(* CODESYS project stec.project

Project tree, tasks and I/O mapping:
  Device : CODESYS Control Win V3, 3S - Smart Software Solutions GmbH, order no. 305021, version 3.5.6.10
    application Application
      libraries: Standard, * (System); Util, * (System)
      task CLP (cyclic, interval t#500ms, priority 1) calls CLP_CONF700
      task executaprocesso (cyclic, interval t#500ms, priority 1) calls Processo
      task RedeFF (cyclic, interval t#500ms, priority 1) calls LD_LT1, LD_LT2, LD_FT1, LD_FT2, LD_FT3, LD_FT4, TT302, FI_01, FI_02
      program CLP_CONF700 [LD]
      global variables CLP_entrada
      global variables CLP_saida
      global variables Var_processo
      function block AI [FBD]
      function block AO [FBD]
      function block PIDCONTROL [FBD]
      program LD_LT1 [FBD]
      function block ALARME [LD]
      program Processo [ST]
      Symbols
      program LD_LT2 [FBD]
      program LD_FT1 [FBD]
      program LD_FT2 [FBD]
      program LD_FT3 [FBD]
      program LD_FT4 [FBD]
      program FI_01 [FBD]
      program TT302 [FBD]
      program FI_02 [FBD]
      global variables Par_processo
      function block ControladorPID [ST]
*)

// Device/Application/CLP_entrada
VAR_GLOBAL
HI_LEVEL01	:BOOL;   // indicação de nivel alto no TAQ
HI_LEVEL02	:BOOL;   // indicação de nivel alto no TP
HI_TEMP01	:BOOL;   // indicação de temperatura alta no TAQ
HI_TEMP02	:BOOL;   // indicação de temperatura altra no TP
HI_FLOW01	:BOOL;   // Indicação de vazão alta na saída do TP
LO_LEVEL01	:BOOL;   // indicação de nivel baixo no TAQ
LO_LEVEL02	:BOOL;   //indicação de nivel baixo no TP

// considere que 01 é TAQ e 02 é TP
END_VAR

// Device/Application/CLP_saida
VAR_GLOBAL
B02	:BOOL;  //comando para ligar/desligar a bomba 1  entrada TP e TAQ
B01	:BOOL;  //comando para ligar/desligar a bomba 2 saida TP
RES	:BOOL;  // comando para ligar/desligar a resistência
END_VAR

// Device/Application/Var_processo
VAR_GLOBAL
	// variáveis anaógicas de saída do processo
	L_TAQ  :REAL :=0.0;  // nivel do TAQ : LT01
	L_TP   :REAL :=0.0;   // nivel do TP : LT02
	T_TAQ  :REAL :=23.5;  // temperatura medida no TAQ :TT01
	T_TP   :REAL :=23.5;   // Temperatura medida no TP : TT02
	Temp_TAQ  :REAL :=23.5;  // temperatura real no TAQ :TT01
	Temp_TP   :REAL :=23.5;   // Temperatura real no TP : TT02
	FI_TAQ :REAL:=0.0;   // Vazão de entrada do TAQ : FT01
	FO_TAQ :REAL:=0.0;   // Vazão saida do TAQ  :FT02
	FI_TP :REAL:=0.0;   // Vazão de entrada do TP : FT03
	FO_TP :REAL:=0.0;   // Vazão saida do TP : FT04
	// variáveis anológicas de entrada do processo
	VI_TAQ :REAL;  // comando para vávula FV01 (LCV1) entrada do TAQ 
	VO_TAQ :REAL;  // comando para vávula FV02 (TCV1) saida do TAQ
    VI_TP :REAL;   // comando para vávula FV03 (LCV2) entrada do TP
	VO_TP :REAL;  // comando para vávula FV04 (FCV1) saida do TP
	TC_TAQ : REAL; // comando para resistência de aquecimento do TAQ (TTC01)
	// variáveis de interface com o CLP
	
END_VAR

// Device/Application/Par_processo
VAR_GLOBAL
	// valores de parametrização do nivel do TAQ
LTAQMAX: REAL := 500.0; // Nível máximo do TAQ
LTAQMIN: REAL :=0.0;   // Nivel minimo do TAQ
LSHTAQ:REAL :=450.0;  // Limite para alarme de nível alto
LSLTAQ:REAL :=60.0;   // Limite para alarme de nível baixo

	//valores de parametrização do nivel do TP
LTPMAX: REAL := 700.0; // Nível máximo do TP
LTPMIN: REAL :=0.0;   // Nivel minimo do TP
LSHTP:REAL :=650.0;  // Limite para alarme de nível alto
LSLTP:REAL :=50.0;   // Limite para alarme de nível baixo

//valores de parametrização da tempearatura do TAQ
TSHTAQ:REAL :=80.0;  // Limite para alarme de temperatura alta alto
TTPMAX: REAL := 100.0;//Temperatura máxima para o TP
TTPMIN: REAL :=0.0;   // Temperatura minima para o TP

//valores de parametrização da tempearatura do TP
TTAQMAX: REAL := 100.0;//Temperatura máxima para o TAQ
TTAQMIN: REAL :=0.0;   // Temperatura minima para o TAQ
TSHTP:REAL :=50.0;  // Limite para alarme de temperatura alta alto

//valores de parametrização da vazao entrada TAQ
FIXTAQ :REAL :=44.0;   // vazão máxima de entrada do TAQ
FIITAQ :REAL :=0.0;     // vazão mínima de entrada do TAQ

//valores de parametrização da vazão saida TAQ
FOXTAQ :REAL :=9.0;   // vazão máxima de saida do TAQ
FOITAQ :REAL :=0.0;     // vazão mínima de saida do TAQ

//valores de parametrização da vazão entrada TP
FIXTP :REAL :=34.0;   // vazão máxima de entrada do TP
FIITP :REAL :=0.0;     // vazão mínima de entrada do TP

//valores de parametrização da vazão saida TP
FOXTP :REAL :=56.0;   // vazão máxima de saida do TP
FOITP :REAL :=0.0;    // vazão mínima de saida do TP
FSH4:REAL :=57.0;  // Limite para alarme de nível alto


//valores de parametrização da potência da resistência de aquecimento do TAQ
PMAX:REAL:=12000;
Temp_Reservatorio:REAL:=23;

DELTAT:REAL:=0.5;     // intervalode de amostragem deve corresponder ao tempo de ciclo da tarefa

END_VAR

// Device/Application/CLP_CONF700
PROGRAM CLP_CONF700
VAR
 
SHB02	:BOOL;   // cahve de software via SCADA para ligar a bomba 2
SHB01	:BOOL;   // cahve de software via SCADA para ligar a bomba 1
SHRES	:BOOL;   // cahve de software via SCADA para ligar a resistência
END_VAR

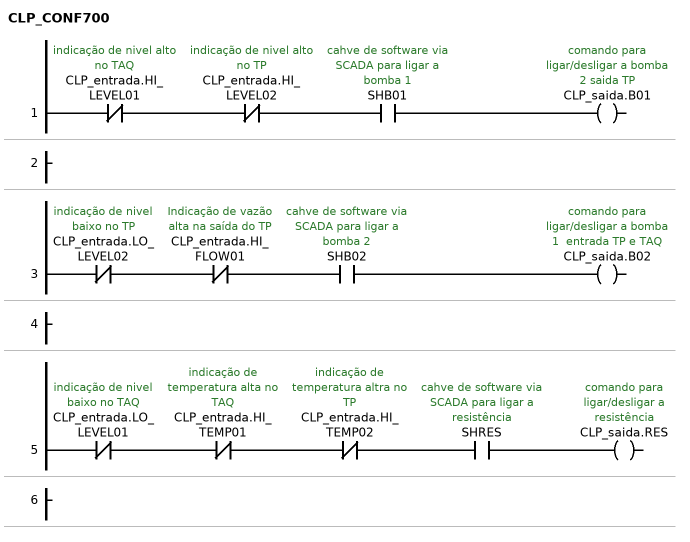
// NETWORK 1
//   CLP_entrada.HI_LEVEL01: indicação de nivel alto no TAQ
//   CLP_entrada.HI_LEVEL02: indicação de nivel alto no TP
//   SHB01: cahve de software via SCADA para ligar a bomba 1
//   CLP_saida.B01: comando para ligar/desligar a bomba 2 saida TP
CLP_saida.B01 := NOT CLP_entrada.HI_LEVEL01 AND NOT CLP_entrada.HI_LEVEL02 AND SHB01;

// NETWORK 2

// NETWORK 3
//   CLP_entrada.LO_LEVEL02: indicação de nivel baixo no TP
//   CLP_entrada.HI_FLOW01: Indicação de vazão alta na saída do TP
//   SHB02: cahve de software via SCADA para ligar a bomba 2
//   CLP_saida.B02: comando para ligar/desligar a bomba 1 entrada TP e TAQ
CLP_saida.B02 := NOT CLP_entrada.LO_LEVEL02 AND NOT CLP_entrada.HI_FLOW01 AND SHB02;

// NETWORK 4

// NETWORK 5
//   CLP_entrada.LO_LEVEL01: indicação de nivel baixo no TAQ
//   CLP_entrada.HI_TEMP01: indicação de temperatura alta no TAQ
//   CLP_entrada.HI_TEMP02: indicação de temperatura altra no TP
//   SHRES: cahve de software via SCADA para ligar a resistência
//   CLP_saida.RES: comando para ligar/desligar a resistência
CLP_saida.RES := NOT CLP_entrada.LO_LEVEL01 AND NOT CLP_entrada.HI_TEMP01 AND NOT CLP_entrada.HI_TEMP02 AND SHRES;

// NETWORK 6

END_PROGRAM

// Device/Application/Processo
PROGRAM Processo
VAR
BETA:REAL:=0.7;   // valor do filtro das vazões
offset:REAL:=23.4;  //  temperatura inicial
cont:INT;         //contador de atrasos
// parametros vazão entrada ATQ
KITAQ:REAL :=  0.73;        // ganho vazão entrada TAQ
ATITAQ:REAL := 4.0;     //  atraso em segundos vazão entrada TAQ
VIATAQ : ARRAY [1..10] OF REAL := [0,0,0,0,0,0,0,0,0,0];  // vetor com valores anteriores da valvula de entrada TAQ
FIATAQ : REAL;  // valor anterior da vazaão de entrada TAQ
KOTAQ:REAL :=  0.128;        // ganho vazão saida TAQ
ATOTAQ:REAL := 4.0;     //  atraso em segundos vazão saida TAQ
VOATAQ : ARRAY [1..10] OF REAL := [0,0,0,0,0,0,0,0,0,0];  // vetor com valores anteriores da valvula saida TAQ
FOATAQ : REAL;  // valor anterior da vazaão de saida TAQ
// parametro para as vazões do TP

KITP:REAL :=  0.68;        // ganho vazão entrada TP
ATITP:REAL := 4.0;     //  atraso em segundos vazão entrada TP
VIATP : ARRAY [1..10] OF REAL := [0,0,0,0,0,0,0,0,0,0];  // vetor com valores anteriores da valvula entrada TAQ
FIATP : REAL;  // valor anterior da vazaão de entrada TP
KOTP :REAL := 0.8;  // ganho vazão saida TP
ATOTP:REAL := 3.0;     //  atraso em segundos vazão saida TP
VOATP : ARRAY [1..10] OF REAL := [0,0,0,0,0,0,0,0,0,0];  // vetor com valores anteriores da valvula saida TAQ
FOATP : REAL;  // valor anterior da vazaão de saida TP
VAZAOTP: REAL;  // variável auxiliar para calcula vazao saida TP
// parametro para valvulas do TAQ
VIXTAQ :REAL :=70.0;   // limite superior de saturação para a vazão máxima valvula entrada TAQ
VIITAQ :REAL :=10.0;     // limite inferior de saturação para a vazão máxima valvula entrada TAQ
VOXTAQ :REAL :=90.0;   // limite superior de saturação para a vazão máxima valvula saida TAQ
VOITAQ :REAL :=20.0;     // limite inferior de saturação para a vazão máxima valvula saida TAQ

// parametro para valvulas do TP
VIXTP :REAL :=60.0;   // limite superior de saturação para a vazão máxima valvula entrada TP
VIITP :REAL :=10.0;     // limite inferior de saturação para a vazão máxima valvula entrada TP
VOXTP :REAL :=80.0;   // limite superior de saturação para a vazão máxima valvula saida TP
VOITP :REAL :=10.0;     // limite inferior de saturação para a vazão máxima valvula saida TP

// parametros para caluclo dos nivies
AREA:REAL:=1.140E5;   // Area dos tanques em mm
CONV:REAL:=16.67E3;  //conversaço de l/min para mm3/s
LATAQ:REAL;    // valor anterior do nivel do TAQ
LATP:REAL;    // valor anterior do nivel do TP
VAZAO:REAL;   // variável auxiliar para calculo do balanço da vazão

Temp_TAQ:REAL;
Temp_TP:REAL;
Vol_TP:REAL;
Vol_TAQ:REAL;

//parametros calculo temperatura TAQ

nataq:REAL:=0.9568E-3;   //numerador discreto função de aquecimento do TAQ
dataq:REAL:=-0.999;   //denominador discreto função de aquecimento do TAQ
nftaq:REAL:=0.0102;   //numerador discreto entrada agua fria no TAQ
dftaq:REAL:=-0.9876;   //denominador discreto entrada agua fria no TAQ
uataq:REAL:=0;    // sinal de entrada para aquecimento do TAQ
sataq:REAL:=0;    // parcela da temperatura de aquecimento do TAQ
U1TAQ : ARRAY [1..50] OF REAL := [0,0,0,0,0,0,0,0,0,0,0,0,0,0,0,0,0,0,0,0,0,0,0,0,0,0,0,0,0,0,0,0,0,0,0,0,0,0,0,0,0,0,0,0,0,0,0,0,0,0]; 
uftaq:REAL:=0;    // sinal de entrada para esfriar o  TAQ
sftaq:REAL:=0;    // parcela da temperatura do esfriamento do TAQ
U2TAQ :ARRAY [1..10] OF REAL :=[0,0,0,0,0,0,0,0,0,0];
Ttaq:REAL;    // auxiliar para somar as parcelas da temperatura e saturar entre offset e 100
potencia:REAL:=0; // auxiliar para potencia como liga/desliga da temperatura
antsf:REAL:=0;  //valor anterior da parcela de resfriamento da temperatura
antsa:REAL:=0; // valor anterior da parcela de aquecimento da temperatura
//parametros calculo temperatura TP

natp:REAL:=0.6297E-3;   //numerador discreto função de aquecimento do TP
datp:REAL:=-0.9967;   //denominador discreto função de aquecimento do TP
nftp:REAL:=0.4225E-4;   //numerador discreto entrada agua fria no TP
dftp:REAL:=-0.9850;   //denominador discreto entrada agua fria no TP
uatp:REAL;    // sinal de entrada para aquecimento do TP
satp:REAL;    // parcela da temperatura de aquecimento do TP
U1TP : ARRAY [1..50] OF REAL := [0,0,0,0,0,0,0,0,0,0,0,0,0,0,0,0,0,0,0,0,0,0,0,0,0,0,0,0,0,0,0,0,0,0,0,0,0,0,0,0,0,0,0,0,0,0,0,0,0,0]; 
uftp:REAL;    // sinal de entrada para esfriar o  TP
sftp:REAL;    // parcela da temperatura do esfriamento do TP
U2TP :ARRAY [1..10] OF REAL :=[0,0,0,0,0,0,0,0,0,0];
Ttp:REAL;    // auxiliar para somar as parcelas da temperatura e saturar entre offset e 100
antpsf:REAL:=0;  //valor anterior da parcela de resfriamento da temperatura
antpsa:REAL:=0; // valor anterior da parcela de aquecimento da temperatura
haux, taux, faux:REAL:=0;  // variaveis auxiliaroes
lixo:REAL:=0;
END_VAR

// atualiza os valores anteriores  das vazões
FIATAQ:=Var_processo.FI_TAQ;
FOATAQ:=Var_processo.FO_TAQ;
FIATP:=Var_processo.FI_TP;
FOATP:=Var_processo.FO_TP;
// atualiza os valores anteriores dos niveis
LATAQ:=Var_processo.L_TAQ;
LATP:=Var_processo.L_TP;
// atualiza os valores anteriores das valvulas  e  dos sinais da temperatura
FOR cont:=10 TO 2 BY -1 DO
		VIATAQ[cont]:=VIATAQ[cont-1]; 
		VOATAQ[cont]:=VOATAQ[cont-1]; 
		VIATP[cont]:=VIATP[cont-1]; 
		VOATP[cont]:=VOATP[cont-1]; 
		U2TAQ[cont]:=U2TAQ[cont-1];
		U2TP[cont]:=U2TP[cont-1];
END_FOR
FOR cont:=50 TO 2 BY -1 DO
		U1TAQ[cont]:=U1TAQ[cont-1];
		U1TP[cont]:=U1TP[cont-1];
END_FOR
// garante a saturação das valvulas entre 0 e 100%
IF Var_processo.VI_TAQ < 0.0
	THEN Var_processo.VI_TAQ:=0.0;
END_IF
IF Var_processo.VI_TAQ > 100.0
	THEN Var_processo.VI_TAQ:=100.0;
END_IF

IF Var_processo.VO_TAQ < 0.0
	THEN Var_processo.VO_TAQ:=0.0;
END_IF
IF Var_processo.VO_TAQ > 100.0
	THEN Var_processo.VO_TAQ:=100.0;
END_IF

IF Var_processo.VI_TP < 0.0
	THEN Var_processo.VI_TP:=0.0;
END_IF
IF Var_processo.VI_TP > 100.0
	THEN Var_processo.VI_TP:=100.0;
END_IF

IF Var_processo.VO_TP < 0.0
	THEN Var_processo.VO_TP:=0.0;
END_IF
IF Var_processo.VO_TP > 100.0
	THEN Var_processo.VO_TP:=100.0;
END_IF

// atualiza a posição mais recente dos vetores de atraso das valvulas
VIATAQ[1]:= Var_processo.VI_TAQ;
VOATAQ[1]:= Var_processo.VO_TAQ;
VIATP[1]:= Var_processo.VI_TP;
VOATP[1]:= Var_processo.VO_TP;

// vazão de entrada do TAQ
Var_processo.FI_TAQ:= MIN(0.7*VIATAQ[8],12/(0.5+EXP(-0.125*(VIATAQ[8]-20))));
IF NOT(CLP_saida.B01) // verifica se a bomba está desligada
	THEN Var_processo.FI_TAQ:=0.0;
END_IF
// dinamica da válvula
Var_processo.FI_TAQ:= BETA*Var_processo.FI_TAQ + (1-BETA)*FIATAQ;

// vazão de saida do TAQ
Var_processo.FO_TAQ:=  SQRT(LATAQ/LTAQMAX*2)*MIN(0.2*VOATAQ[8],7.2/(0.8+EXP(-0.1125*(VOATAQ[8]-50)))); 

// dinamica valvula
Var_processo.FO_TAQ:= BETA*Var_processo.FO_TAQ + (1-BETA)*FOATAQ;

// vazão de entrada do TP
Var_processo.FI_TP:=  MIN(1.0*VIATP[8],25.85/(0.615+EXP(-0.1*(VIATP[8]-35))));
IF NOT(CLP_saida.B01) // verifica se a bomba está desligada
	THEN Var_processo.FI_TP:=0.0;
END_IF
 
// coloca um filtro para a mudança não ser muito brusca
Var_processo.FI_TP:= BETA*Var_processo.FI_TP + (1-BETA)*FIATP;

// vazão de saida do TP
//é preciso uma variável auxiliar para evitar que o alarme dispare antes do calculo completo da vazão
VAZAOTP:=  MIN(1.3*VOATP[8],53/(0.964+EXP(-0.097*(VOATP[8]-35))));
IF NOT(CLP_saida.B02) // verifica se a bomba está desligada
	THEN VAZAOTP:=0.0;
END_IF

// dinamica valvula

Var_processo.FO_TP:= BETA*VAZAOTP + (1-BETA)*FOATP;

// calcula os niveis pelo balançco dinamico das vazões
//Nivel do TAQ
VAZAO:=Var_processo.FI_TAQ-Var_processo.FO_TAQ;
VAZAO:=VAZAO*CONV;
Var_processo.L_TAQ:= LATAQ+(VAZAO*DELTAT)/AREA;
IF Var_processo.L_TAQ  < 0.0
	THEN Var_processo.L_TAQ:=0.0;
END_IF
IF Var_processo.L_TAQ > LTAQMAX
	THEN Var_processo.L_TAQ:=LTAQMAX;
END_IF

//Nivel do TP
VAZAO:=Var_processo.FI_TP + Var_processo.FO_TAQ - Var_processo.FO_TP ;
VAZAO:=VAZAO*CONV;
Var_processo.L_TP:= LATP+(VAZAO*DELTAT)/AREA;
IF Var_processo.L_TP  < 0.0
	THEN Var_processo.L_TP:=0.0;
END_IF
IF Var_processo.L_TP > LTPMAX
	THEN Var_processo.L_TP:=LTPMAX;
END_IF

//calculo das temperaturas pelos modelos pelo balanço de massa e energia
//Temperatura do TAQ parcela de aquecimento
IF CLP_saida.RES
	THEN potencia:=Par_processo.PMAX *(Var_processo.TC_TAQ/100+SIN(2*(1-Var_processo.TC_TAQ/100)*3.1416)/(2*3.1416));//(pi-theta)/2 + sin(2theta)/4
	ELSE potencia:=0;
END_IF

Vol_TAQ:=AREA*LATAQ*1E-6+DELTAT*(FIATAQ-FOATAQ)/60;
IF Vol_TAQ<=0
	THEN Vol_TAQ:=1E-2;
END_IF

Temp_TAQ:=Var_processo.Temp_TAQ+potencia*DELTAT/4200/Vol_TAQ;
Temp_TAQ:=Temp_TAQ+FIATAQ*DELTAT/60/Vol_TAQ*(Par_processo.Temp_Reservatorio-Var_processo.Temp_TAQ);

U1TAQ[1]:=Temp_TAQ;   // atualiza a  posição mais recente do vetor de atrasos
Var_processo.T_TAQ := Var_processo.T_TAQ +BETA * (U1TAQ[50]-Var_processo.T_TAQ); 

//Temperatura do TP
//--------------------------------------------------------------
Vol_TP:=AREA*LATP*1E-6+DELTAT*(FIATP+FOATAQ-FOATP)/60;
IF Vol_TP<=0
	THEN Vol_TP:=1E-2;
END_IF

Temp_TP:=Var_processo.Temp_TP+DELTAT*FIATP/60/Vol_TP*(Par_processo.Temp_Reservatorio-Var_processo.Temp_TP);
Temp_TP:=Temp_TP+DELTAT*FOATAQ/60/Vol_TP*(Var_processo.Temp_TAQ-Var_processo.Temp_TP);

U1TP[1]:=Temp_TP;   // atualiza a  posição mais recente do vetor de atrasos
Var_processo.T_TP := Var_processo.T_TP + BETA*(U1TP[50]-Var_processo.T_TP); 

Var_processo.Temp_TAQ:=Temp_TAQ;
Var_processo.Temp_TP:=Temp_TP;

END_PROGRAM

// Device/Application/ALARME
FUNCTION_BLOCK ALARME
VAR_INPUT
	Valor:REAL;  // valor atual da variável
	Limite: REAL;  // Limite para setar o alarme
	Posicao: BOOL;  // Posição do alarme ALTO=1  Baixo = 0
END_VAR
VAR_OUTPUT
	SETALARME: BOOL; // Indica condição verdadira se ocorrência de alarme
END_VAR

VAR
ASH,ASL:BOOL;    	
END_VAR

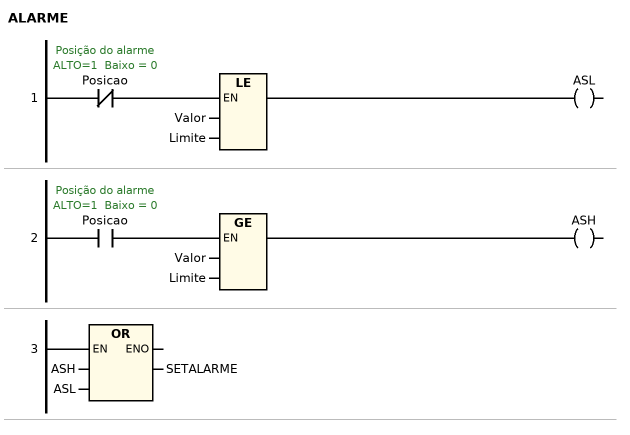
// NETWORK 1
//   Posicao: Posição do alarme ALTO=1 Baixo = 0
//   Valor: valor atual da variável
//   Limite: Limite para setar o alarme
ASL := NOT Posicao AND Valor <= Limite;

// NETWORK 2
//   Posicao: Posição do alarme ALTO=1 Baixo = 0
//   Valor: valor atual da variável
//   Limite: Limite para setar o alarme
ASH := Posicao AND Valor >= Limite;

// NETWORK 3
//   SETALARME: Indica condição verdadira se ocorrência de alarme
SETALARME := ASH OR ASL;

END_FUNCTION_BLOCK

// Device/Application/LD_LT1
// Corresponde ao instrumento LD-302 Medidor e controlador do Nivel do TAQ
PROGRAM LD_LT1
VAR
ModoNivelTAQ	:BOOL :=TRUE;	//	modo PID nivel TAQ
SetPointNivelTAQ	:REAL:=0.0;	//	Set point PID nivel TAQ
ValorManualNivelTAQ	:REAL:=0.0;	//	Valor manaual PID nivel TAQ
PVNivelTAQ	:REAL;	//	Valor entrada PID nivel TAQ
GanhoNivelTAQ	:REAL:=1.0;	//	Ganho PID nivel TAQ
GanhoFF 		:REAL:= Var_processo.FO_TAQ*0.375;
TINivelTAQ	:REAL:=10.0;	//	Ti PID nivel TAQ
TDNivelTAQ	:REAL:=0.0;	//	Td PID nivel TAQ

STPIDLT1:BOOL;      // inidicação de saturação na MV
OVPIDLT1:BOOL;      // indicação de overflow no termo integral

LCV1	:REAL;	//	comando de abertura da Valvula LCV1 que controla o nive do TAQ
LT01    :REAL;  // Nivel do TAQ
DIST	:REAL;  // Disturbio no 
AILT1: AI;   //Bloco de entrada analógica
PIDLT1: PIDCONTROL;  //Bloco PID
ALHLT1: ALARME;    //Bloco de Alarme ALTO
ALLLT1: ALARME;     //Bloco de Alarme Baixo
END_VAR

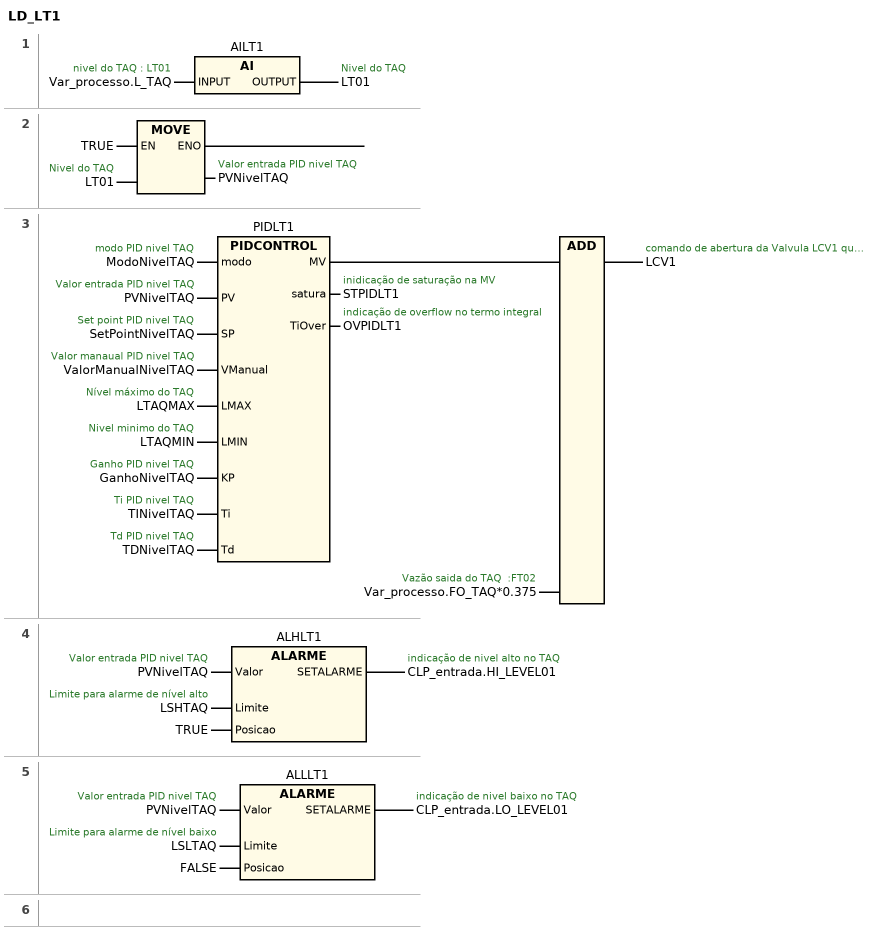
// NETWORK 1
//   AILT1: Bloco de entrada analógica
//   Var_processo.L_TAQ: nivel do TAQ : LT01
//   LT01: Nivel do TAQ
AILT1(INPUT := Var_processo.L_TAQ); // AI
LT01 := AILT1.OUTPUT;

// NETWORK 2
//   LT01: Nivel do TAQ
//   PVNivelTAQ: Valor entrada PID nivel TAQ
PVNivelTAQ := LT01;

// NETWORK 3
//   PIDLT1: Bloco PID
//   ModoNivelTAQ: modo PID nivel TAQ
//   PVNivelTAQ: Valor entrada PID nivel TAQ
//   SetPointNivelTAQ: Set point PID nivel TAQ
//   ValorManualNivelTAQ: Valor manaual PID nivel TAQ
//   LTAQMAX: Nível máximo do TAQ
//   LTAQMIN: Nivel minimo do TAQ
//   GanhoNivelTAQ: Ganho PID nivel TAQ
//   TINivelTAQ: Ti PID nivel TAQ
//   TDNivelTAQ: Td PID nivel TAQ
//   STPIDLT1: inidicação de saturação na MV
//   OVPIDLT1: indicação de overflow no termo integral
//   Var_processo.FO_TAQ*0.375: Vazão saida do TAQ :FT02
//   LCV1: comando de abertura da Valvula LCV1 que controla o nive do TAQ
PIDLT1(
    modo := ModoNivelTAQ,
    PV := PVNivelTAQ,
    SP := SetPointNivelTAQ,
    VManual := ValorManualNivelTAQ,
    LMAX := LTAQMAX,
    LMIN := LTAQMIN,
    KP := GanhoNivelTAQ,
    Ti := TINivelTAQ,
    Td := TDNivelTAQ,
    satura => STPIDLT1,
    TiOver => OVPIDLT1); // PIDCONTROL
LCV1 := PIDLT1.MV + (Var_processo.FO_TAQ*0.375);

// NETWORK 4
//   ALHLT1: Bloco de Alarme ALTO
//   PVNivelTAQ: Valor entrada PID nivel TAQ
//   LSHTAQ: Limite para alarme de nível alto
//   CLP_entrada.HI_LEVEL01: indicação de nivel alto no TAQ
ALHLT1(Valor := PVNivelTAQ, Limite := LSHTAQ, Posicao := TRUE); // ALARME
CLP_entrada.HI_LEVEL01 := ALHLT1.SETALARME;

// NETWORK 5
//   ALLLT1: Bloco de Alarme Baixo
//   PVNivelTAQ: Valor entrada PID nivel TAQ
//   LSLTAQ: Limite para alarme de nível baixo
//   CLP_entrada.LO_LEVEL01: indicação de nivel baixo no TAQ
ALLLT1(Valor := PVNivelTAQ, Limite := LSLTAQ, Posicao := FALSE); // ALARME
CLP_entrada.LO_LEVEL01 := ALLLT1.SETALARME;

// NETWORK 6

END_PROGRAM

// Device/Application/AI
FUNCTION_BLOCK AI
// represneta o bloco AI da rede FF responsável por obter uma variável analógica do processo
// disponibilizar a variável em unidade de engenharia para a rede FF 
VAR_INPUT
	INPUT:REAL;  // variável analógiva de entrada do processo
END_VAR
VAR_OUTPUT
	OUTPUT :REAL;  // variável para a rede FF
END_VAR

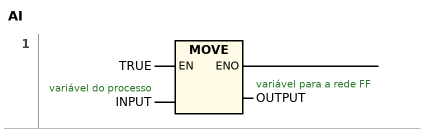
// NETWORK 1
//   INPUT: variável do processo
//   OUTPUT: variável para a rede FF
OUTPUT := INPUT;

END_FUNCTION_BLOCK

// Device/Application/PIDCONTROL
FUNCTION_BLOCK PIDCONTROL
VAR_INPUT
	modo : BOOL;  // modo de operação da malha de controle  Manual=1  Automatico=0
	PV    :REAL;  // variável de processo (entrada do PID)
	SP   : REAL;  // valor de referência para a malha fechada
	LMAX:  REAL;  // Limite superior da PV;
	LMIN: REAL;   // Limite inferiro da PV;
	KP : REAL; // ganho do controlador
	Ti :REAL;   // tempo integral em segundos
	Td  :REAL;  //Tempo derivativo em segundos
END_VAR
VAR_OUTPUT
	MV    :REAL;  // variável manipulada (saida do PID)
	satura : BOOL; // variável indicativa que houve saturação da MV
	TiOver:  BOOL;  // vafiável indicativa que houve saturação do termo integral
END_VAR

VAR_IN_OUT
	VManual : REAL;  // valor de referência para a saida do controlador quando em modo manual	
END_VAR

VAR
	controlador: PID;  ///bloco genério PID Y(s)= KP(1+ (1/sTi) + sTd)E(s)
	controlePID: ControladorPID;
END_VAR

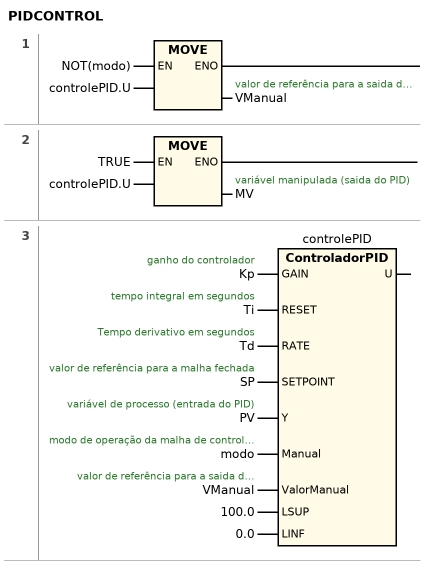
// NETWORK 1
//   VManual: valor de referência para a saida do controlador quando em modo manual
IF NOT(modo) THEN VManual := controlePID.U; END_IF

// NETWORK 2
//   MV: variável manipulada (saida do PID)
MV := controlePID.U;

// NETWORK 3
//   controlePID: bloco genério PID Y(s)= KP(1+ (1/sTi) + sTd)E(s)
//   Kp: ganho do controlador
//   Ti: tempo integral em segundos
//   Td: Tempo derivativo em segundos
//   SP: valor de referência para a malha fechada
//   PV: variável de processo (entrada do PID)
//   modo: modo de operação da malha de controle Manual=1 Automatico=0
//   VManual: valor de referência para a saida do controlador quando em modo manual
controlePID(
    GAIN := Kp,
    RESET := Ti,
    RATE := Td,
    SETPOINT := SP,
    Y := PV,
    Manual := modo,
    ValorManual := VManual,
    LSUP := 100.0,
    LINF := 0.0); // ControladorPID

END_FUNCTION_BLOCK

// Device/Application/ControladorPID
FUNCTION_BLOCK ControladorPID
VAR_INPUT
	GAIN: REAL;
	RESET: REAL;
	RATE: REAL;
	SETPOINT: REAL := 0.0;
	Y: REAL;
	Manual: BOOL := FALSE;
	ValorManual: REAL;
	LSUP: REAL;
	LINF: REAL;
END_VAR
VAR_OUTPUT
	U: REAL := LINF;
END_VAR
VAR
	Kp: REAL;
	BETA: REAL;
	GAMMA: REAL;
	Kd: REAL;
	Aux2: REAL;
	Aux: REAL := 0.0;
	PI: REAL := LINF;
	D: REAL := 0.0;
	Yant: REAL := 0.0;
END_VAR

VAR CONSTANT
	ALPHA: REAL := 0.13;
END_VAR


Kp:=GAIN*(1+DELTAT/(2*RESET));
BETA:=2*DELTAT/(2*RESET+DELTAT);
GAMMA:=1/(1+ALPHA*RATE/DELTAT);
Kd:=GAIN*RATE/DELTAT;
Aux2 := Kp*(SETPOINT-Y)+Aux;
Aux:= (1-BETA) * Aux + BETA*PI;
D := (1-GAMMA)*D+GAMMA*Kd*(Yant-Y);
Yant:=Y;
PI:=Aux2;
IF (Manual)
THEN U:= ValorManual;
ELSE U:=PI+D;
END_IF

IF (U>LSUP)
THEN U:=LSUP;
END_IF
IF (U<LINF)
THEN U:=LINF;
END_IF
PI:=U-D;

END_FUNCTION_BLOCK

// Device/Application/AO
FUNCTION_BLOCK AO
// represneta o bloco AO da rede FF responsável por enviar uma variável analogica da rede FF e
// enviar a variável para o processo 
VAR_INPUT
	INPUT: REAL; // variavel da rede FF
END_VAR
VAR_OUTPUT
	OUTPUT :REAL; // variável do processo
END_VAR
VAR
END_VAR

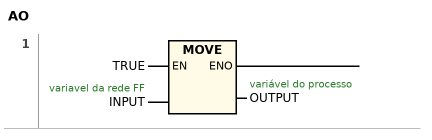
// NETWORK 1
//   INPUT: variavel da rede FF
//   OUTPUT: variável do processo
OUTPUT := INPUT;

END_FUNCTION_BLOCK

// Device/Application/LD_LT2
// Corresponde ao instrumento LD-302 Medidor e controlador do Nivel do TP
PROGRAM LD_LT2
VAR
ModoNivelTP	:BOOL :=TRUE;	//	modo PID nivel TP
SetPointNivelTP	:REAL;	//	Set point PID nivel TP
ValorManualNivelTP	:REAL:=0.0;	//	Valor manaual PID nivel TP
PVNivelTP	:REAL;	//	Valor entrada PID nivel TP
GanhoNivelTP	:REAL:=1.0;	//	Ganho PID nivel TP
TINivelTP	:REAL:=10.0;	//	Ti PID nivel TP
TDNivelTP	:REAL:=0.0;	//	Td PID nivel TP



STPIDLT2:BOOL;      // inidicação de saturação na MV
OVPIDLT2:BOOL;      // indicação de overflow no termo integral

LCV2	:REAL;	//	comando de abertura da Valvula LCV1 que controla o nive do TAQ
LT02    :REAL;  // nivel do TP
AILT2: AI;   //Bloco de entrada analógica
AOLT2: AO;   //Bloco de saída analógica
PIDLT2: PIDCONTROL;  //Bloco PID
ALHLT2: ALARME;    //Bloco de Alarme ALTO
ALLLT2: ALARME;     //Bloco de Alarme Baixo
END_VAR

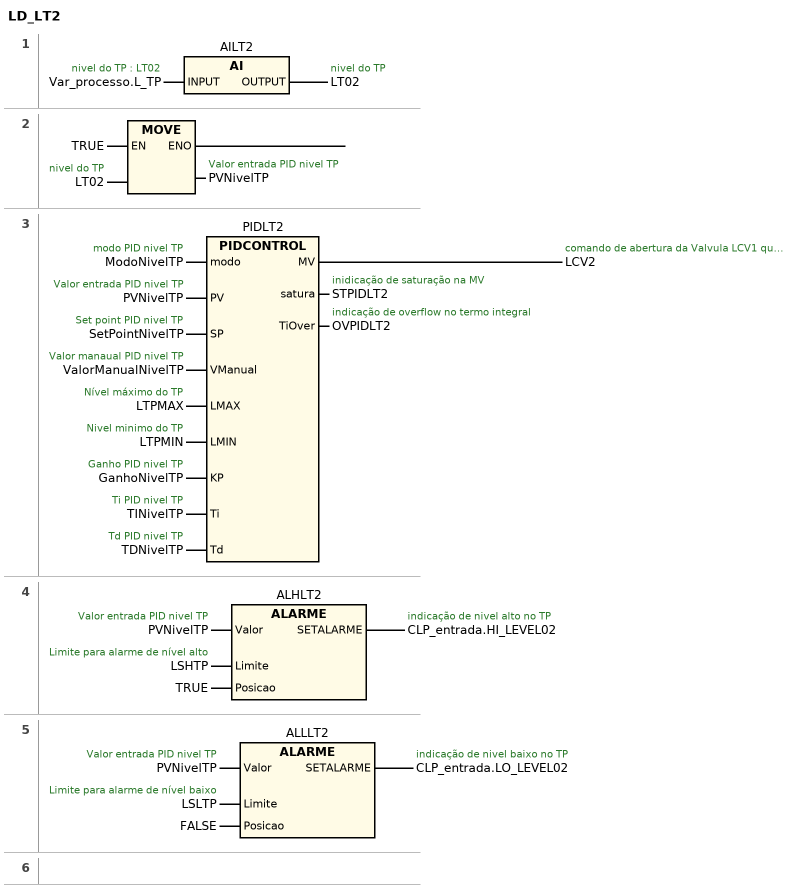
// NETWORK 1
//   AILT2: Bloco de entrada analógica
//   Var_processo.L_TP: nivel do TP : LT02
//   LT02: nivel do TP
AILT2(INPUT := Var_processo.L_TP); // AI
LT02 := AILT2.OUTPUT;

// NETWORK 2
//   LT02: nivel do TP
//   PVNivelTP: Valor entrada PID nivel TP
PVNivelTP := LT02;

// NETWORK 3
//   PIDLT2: Bloco PID
//   ModoNivelTP: modo PID nivel TP
//   PVNivelTP: Valor entrada PID nivel TP
//   SetPointNivelTP: Set point PID nivel TP
//   ValorManualNivelTP: Valor manaual PID nivel TP
//   LTPMAX: Nível máximo do TP
//   LTPMIN: Nivel minimo do TP
//   GanhoNivelTP: Ganho PID nivel TP
//   TINivelTP: Ti PID nivel TP
//   TDNivelTP: Td PID nivel TP
//   STPIDLT2: inidicação de saturação na MV
//   OVPIDLT2: indicação de overflow no termo integral
//   LCV2: comando de abertura da Valvula LCV1 que controla o nive do TAQ
PIDLT2(
    modo := ModoNivelTP,
    PV := PVNivelTP,
    SP := SetPointNivelTP,
    VManual := ValorManualNivelTP,
    LMAX := LTPMAX,
    LMIN := LTPMIN,
    KP := GanhoNivelTP,
    Ti := TINivelTP,
    Td := TDNivelTP,
    satura => STPIDLT2,
    TiOver => OVPIDLT2); // PIDCONTROL
LCV2 := PIDLT2.MV;

// NETWORK 4
//   ALHLT2: Bloco de Alarme ALTO
//   PVNivelTP: Valor entrada PID nivel TP
//   LSHTP: Limite para alarme de nível alto
//   CLP_entrada.HI_LEVEL02: indicação de nivel alto no TP
ALHLT2(Valor := PVNivelTP, Limite := LSHTP, Posicao := TRUE); // ALARME
CLP_entrada.HI_LEVEL02 := ALHLT2.SETALARME;

// NETWORK 5
//   ALLLT2: Bloco de Alarme Baixo
//   PVNivelTP: Valor entrada PID nivel TP
//   LSLTP: Limite para alarme de nível baixo
//   CLP_entrada.LO_LEVEL02: indicação de nivel baixo no TP
ALLLT2(Valor := PVNivelTP, Limite := LSLTP, Posicao := FALSE); // ALARME
CLP_entrada.LO_LEVEL02 := ALLLT2.SETALARME;

// NETWORK 6

END_PROGRAM

// Device/Application/LD_FT1
// Corresponde ao instrumento LD-302 Medidor vazão de entrada de agua fria do TAQ
PROGRAM LD_FT1
VAR
	FT1:REAL;  // vazão de entrada do TAQ
	AIFT1: AI;   //Bloco de entrada analógica
END_VAR

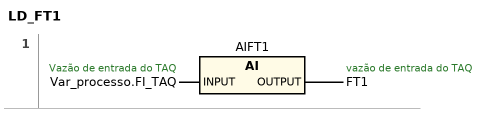
// NETWORK 1
//   AIFT1: Bloco de entrada analógica
//   Var_processo.FI_TAQ: Vazão de entrada do TAQ
//   FT1: vazão de entrada do TAQ
AIFT1(INPUT := Var_processo.FI_TAQ); // AI
FT1 := AIFT1.OUTPUT;

END_PROGRAM

// Device/Application/LD_FT2
// Corresponde ao instrumento LD-302 Medidor vazão de saida do TAQ
// Essa vazão também corresponde a entrada de água quente do TP
PROGRAM LD_FT2
VAR
	FT2:REAL;  // vazão de saida do TAQ
	AIFT2: AI;   //Bloco de entrada analógica
END_VAR

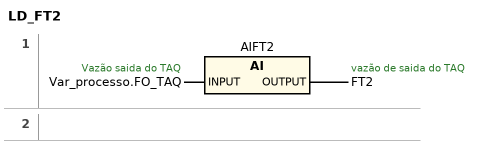
// NETWORK 1
//   AIFT2: Bloco de entrada analógica
//   Var_processo.FO_TAQ: Vazão saida do TAQ
//   FT2: vazão de saida do TAQ
AIFT2(INPUT := Var_processo.FO_TAQ); // AI
FT2 := AIFT2.OUTPUT;

// NETWORK 2

END_PROGRAM

// Device/Application/LD_FT3
// corresponde ao instrumento LD302 medidor de vazão de entrada de água fria no TP
PROGRAM LD_FT3
VAR
	FT3: REAL;  // vazão vazão de entrada de água fria no TP
	AIFT3: AI;   //Bloco de entrada analógica
END_VAR

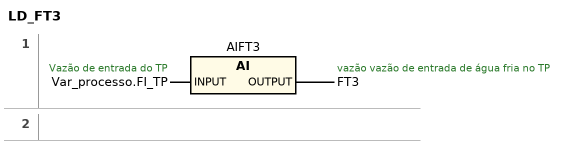
// NETWORK 1
//   AIFT3: Bloco de entrada analógica
//   Var_processo.FI_TP: Vazão de entrada do TP
//   FT3: vazão vazão de entrada de água fria no TP
AIFT3(INPUT := Var_processo.FI_TP); // AI
FT3 := AIFT3.OUTPUT;

// NETWORK 2

END_PROGRAM

// Device/Application/LD_FT4
// Corresponde ao instrumento LD-302 Medidor e controlador de vazão de saida do TP
PROGRAM LD_FT4
VAR
ModoVazaoSaidaTP	:BOOL:=TRUE;	//	modo PID vazão saída TP
SetPointVazaoSaidaTP	:REAL;	//	Set point PID vazão saida TP
ValorManualVazaoSaidaTP	:REAL:=0.0;	//	Valor manual PID vazao saida TP
PVVazaoSaidaTP	:REAL;	//	Valor entrada PID vazao saida TP
GanhoVazaoSaidaTP	:REAL:=1.0;	//	Ganho PID vazão saida TP
TIVazaoSaidaTP	:REAL:=10.0;	//	Ti PID vazao saida TP
TDVazaoSaidaTP	:REAL:=0.0;	//	Td PID vazão saida TP

STPIDFT4: BOOL;      // inidicação de saturação na MV
OVPIDFT4: BOOL;      // indicação de overflow no termo integral

FCV1	:REAL;	//	comando de abertura da Valvula FCV1 que controla a vazão de saida do TP
FT4	    :REAL;  //  vazão de saida do TP
AIFT4: AI;   //Bloco de entrada analógica

PIDFT4: PIDCONTROL;  //Bloco PID
ALHFT4: ALARME;    //Bloco de Alarme ALTO

	
END_VAR

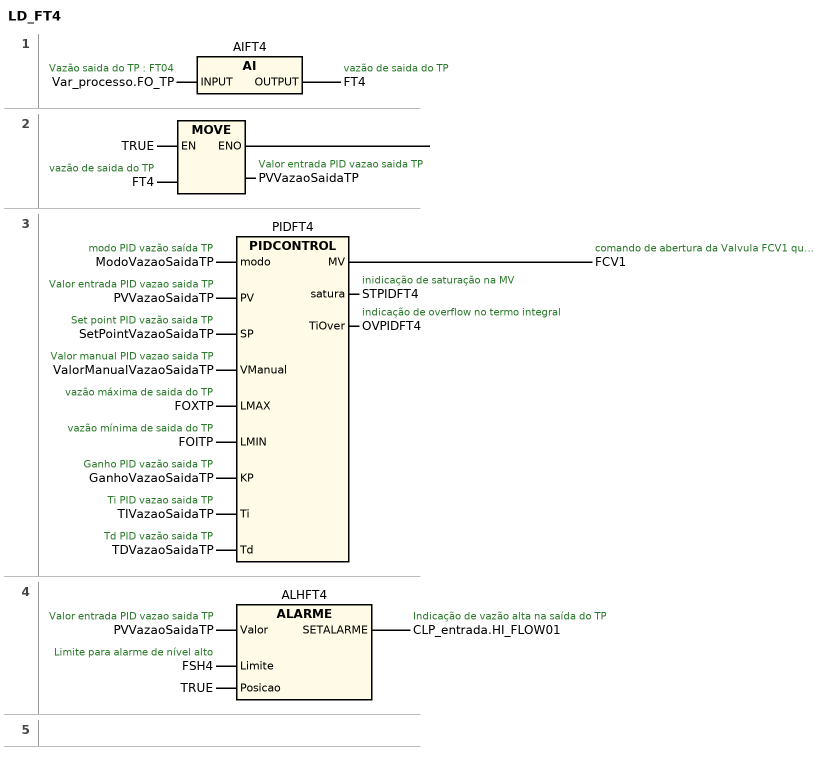
// NETWORK 1
//   AIFT4: Bloco de entrada analógica
//   Var_processo.FO_TP: Vazão saida do TP : FT04
//   FT4: vazão de saida do TP
AIFT4(INPUT := Var_processo.FO_TP); // AI
FT4 := AIFT4.OUTPUT;

// NETWORK 2
//   FT4: vazão de saida do TP
//   PVVazaoSaidaTP: Valor entrada PID vazao saida TP
PVVazaoSaidaTP := FT4;

// NETWORK 3
//   PIDFT4: Bloco PID
//   ModoVazaoSaidaTP: modo PID vazão saída TP
//   PVVazaoSaidaTP: Valor entrada PID vazao saida TP
//   SetPointVazaoSaidaTP: Set point PID vazão saida TP
//   ValorManualVazaoSaidaTP: Valor manual PID vazao saida TP
//   FOXTP: vazão máxima de saida do TP
//   FOITP: vazão mínima de saida do TP
//   GanhoVazaoSaidaTP: Ganho PID vazão saida TP
//   TIVazaoSaidaTP: Ti PID vazao saida TP
//   TDVazaoSaidaTP: Td PID vazão saida TP
//   STPIDFT4: inidicação de saturação na MV
//   OVPIDFT4: indicação de overflow no termo integral
//   FCV1: comando de abertura da Valvula FCV1 que controla a vazão de saida do TP
PIDFT4(
    modo := ModoVazaoSaidaTP,
    PV := PVVazaoSaidaTP,
    SP := SetPointVazaoSaidaTP,
    VManual := ValorManualVazaoSaidaTP,
    LMAX := FOXTP,
    LMIN := FOITP,
    KP := GanhoVazaoSaidaTP,
    Ti := TIVazaoSaidaTP,
    Td := TDVazaoSaidaTP,
    satura => STPIDFT4,
    TiOver => OVPIDFT4); // PIDCONTROL
FCV1 := PIDFT4.MV;

// NETWORK 4
//   ALHFT4: Bloco de Alarme ALTO
//   PVVazaoSaidaTP: Valor entrada PID vazao saida TP
//   FSH4: Limite para alarme de nível alto
//   CLP_entrada.HI_FLOW01: Indicação de vazão alta na saída do TP
ALHFT4(Valor := PVVazaoSaidaTP, Limite := FSH4, Posicao := TRUE); // ALARME
CLP_entrada.HI_FLOW01 := ALHFT4.SETALARME;

// NETWORK 5

END_PROGRAM

// Device/Application/TT302
// Corresponde ao instrumento TT-302 Medidor de temperatura do TAQ 
//e do  medidor/controlador de temperatura do TP
PROGRAM TT302
VAR
ModoTempTP	:BOOL:=TRUE;	//	modo PID temperatura TP
SetPointTempTP	:REAL;	//	Set point PID temperatura TP
ValorManualTempTP	:REAL:=0.0;	//	Valor manual PID temperatura TP
PVTempTP	:REAL;	//	Valor entrada PID temperatura TP
GanhoTempTP	:REAL:=1.0;	//	Ganho PID temperatura TP
TITempTP	:REAL:=10.0;	//	Ti PID temperatura TP
TDTempTP	:REAL:=0.0;	//	Td PID temperatura TP

TCV1	:REAL; // comando de abertura da Valvula TCV1
TT01   : REAL; // temperatura do TAQ
TT02   : REAL; // temperatura do TP


STPIDTT1:BOOL;      // inidicação de saturação na MV
OVPIDTT1:BOOL;      // indicação de overflow no termo integral

// para o TP
AITT2: AI;   //Bloco de entrada analógica
PIDTT2: PIDCONTROL;  //Bloco PID
ALHTT2: ALARME;    //Bloco de Alarme ALTO

// para o TAQ
AITT1: AI;   //Bloco de entrada analógica
ALHTT1: ALARME;    //Bloco de Alarme ALTO

END_VAR

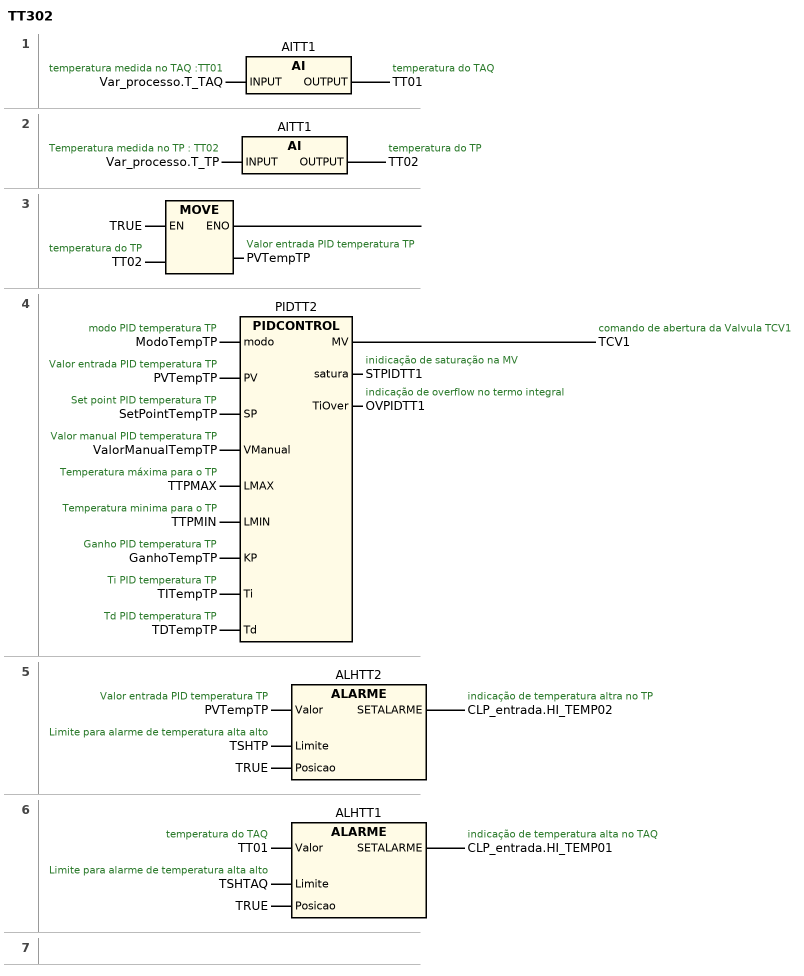
// NETWORK 1
//   AITT1: Bloco de entrada analógica
//   Var_processo.T_TAQ: temperatura medida no TAQ :TT01
//   TT01: temperatura do TAQ
AITT1(INPUT := Var_processo.T_TAQ); // AI
TT01 := AITT1.OUTPUT;

// NETWORK 2
//   AITT1: Bloco de entrada analógica
//   Var_processo.T_TP: Temperatura medida no TP : TT02
//   TT02: temperatura do TP
AITT1(INPUT := Var_processo.T_TP); // AI
TT02 := AITT1.OUTPUT;

// NETWORK 3
//   TT02: temperatura do TP
//   PVTempTP: Valor entrada PID temperatura TP
PVTempTP := TT02;

// NETWORK 4
//   PIDTT2: Bloco PID
//   ModoTempTP: modo PID temperatura TP
//   PVTempTP: Valor entrada PID temperatura TP
//   SetPointTempTP: Set point PID temperatura TP
//   ValorManualTempTP: Valor manual PID temperatura TP
//   TTPMAX: Temperatura máxima para o TP
//   TTPMIN: Temperatura minima para o TP
//   GanhoTempTP: Ganho PID temperatura TP
//   TITempTP: Ti PID temperatura TP
//   TDTempTP: Td PID temperatura TP
//   STPIDTT1: inidicação de saturação na MV
//   OVPIDTT1: indicação de overflow no termo integral
//   TCV1: comando de abertura da Valvula TCV1
PIDTT2(
    modo := ModoTempTP,
    PV := PVTempTP,
    SP := SetPointTempTP,
    VManual := ValorManualTempTP,
    LMAX := TTPMAX,
    LMIN := TTPMIN,
    KP := GanhoTempTP,
    Ti := TITempTP,
    Td := TDTempTP,
    satura => STPIDTT1,
    TiOver => OVPIDTT1); // PIDCONTROL
TCV1 := PIDTT2.MV;

// NETWORK 5
//   ALHTT2: Bloco de Alarme ALTO
//   PVTempTP: Valor entrada PID temperatura TP
//   TSHTP: Limite para alarme de temperatura alta alto
//   CLP_entrada.HI_TEMP02: indicação de temperatura altra no TP
ALHTT2(Valor := PVTempTP, Limite := TSHTP, Posicao := TRUE); // ALARME
CLP_entrada.HI_TEMP02 := ALHTT2.SETALARME;

// NETWORK 6
//   ALHTT1: Bloco de Alarme ALTO
//   TT01: temperatura do TAQ
//   TSHTAQ: Limite para alarme de temperatura alta alto
//   CLP_entrada.HI_TEMP01: indicação de temperatura alta no TAQ
ALHTT1(Valor := TT01, Limite := TSHTAQ, Posicao := TRUE); // ALARME
CLP_entrada.HI_TEMP01 := ALHTT1.SETALARME;

// NETWORK 7

END_PROGRAM

// Device/Application/FI_01
// Corresponde ao instrumento FI302 conversor FF para 4 a 20mA das valvulas TCV1 e FCV1
PROGRAM FI_01
VAR
	AO_01: AO;  // bloco de saida da valvula TCV1 que corresponde a valvula de saida do TAQ
	AO_02 : AO; // bloco de saida do valcvula FCV1 que corresponde a valvula de saida do TP 
	
END_VAR

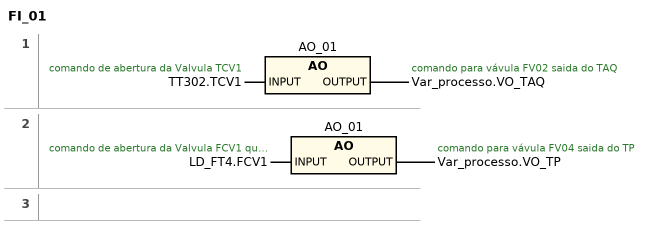
// NETWORK 1
//   TT302.TCV1: comando de abertura da Valvula TCV1
//   Var_processo.VO_TAQ: comando para vávula FV02 saida do TAQ
AO_01(INPUT := TT302.TCV1); // AO
Var_processo.VO_TAQ := AO_01.OUTPUT;

// NETWORK 2
//   AO_01: bloco de saida da valvula TCV1 que corresponde a valvula de saida do TAQ
//   LD_FT4.FCV1: comando de abertura da Valvula FCV1 que controla a vazão de saida do TP
//   Var_processo.VO_TP: comando para vávula FV04 saida do TP
AO_01(INPUT := LD_FT4.FCV1); // AO
Var_processo.VO_TP := AO_01.OUTPUT;

// NETWORK 3

END_PROGRAM

// Device/Application/FI_02
// Corresponde ao instrumento FI302 conversor FF para 4 a 20mA das valvulas TCV1 e FCV1

PROGRAM FI_02
VAR
ModoTempTAQ	:BOOL:=TRUE;	//	modo PID temperatura TAQ
SetPointTempTAQ	:REAL;	//	Set point PID temperatura TAQ
ValorManualTempTAQ	:REAL:=0.0;	//	Valor manual PID temperatura TAQ
PVTempTAQ	:REAL;	//	Valor entrada PID temperatura TAQ
GanhoTempTAQ	:REAL:=1.0;	//	Ganho PID temperatura TAQ
TITempTAQ	:REAL:=10.0;	//	Ti PID temperatura TAQ
TDTempTAQ	:REAL;	//	Td PID temperatura TAQ
TTC01	:REAL;	//	Comando para a resistência do TAQ

STPIDTT1:BOOL;      // inidicação de saturação na MV
OVPIDTT1:BOOL;      // indicação de overflow no termo integral

	AO_01: AO;  // bloco de saida da valvula LCV1 que corresponde a valvula de entrada do TAQ
	AO_02 : AO; // bloco de saida do valcvula LCV2 que corresponde a valvula de entrada do TP 
	AO_03 : AO; // bloco de saida para a resistência de aquecimento
	PIDTT1: PIDCONTROL;  //Bloco PID para controle de temperatura do TAQ
END_VAR

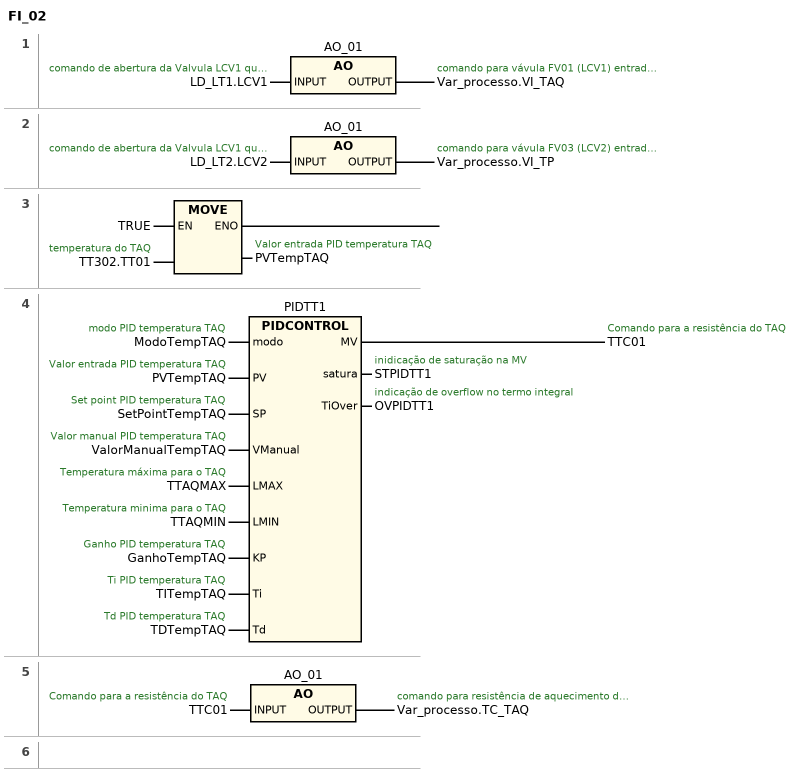
// NETWORK 1
//   AO_01: bloco de saida da valvula LCV1 que corresponde a valvula de entrada do TAQ
//   LD_LT1.LCV1: comando de abertura da Valvula LCV1 que controla o nive do TAQ
//   Var_processo.VI_TAQ: comando para vávula FV01 (LCV1) entrada do TAQ
AO_01(INPUT := LD_LT1.LCV1); // AO
Var_processo.VI_TAQ := AO_01.OUTPUT;

// NETWORK 2
//   AO_01: bloco de saida da valvula LCV1 que corresponde a valvula de entrada do TAQ
//   LD_LT2.LCV2: comando de abertura da Valvula LCV1 que controla o nive do TAQ
//   Var_processo.VI_TP: comando para vávula FV03 (LCV2) entrada do TP
AO_01(INPUT := LD_LT2.LCV2); // AO
Var_processo.VI_TP := AO_01.OUTPUT;

// NETWORK 3
//   TT302.TT01: temperatura do TAQ
//   PVTempTAQ: Valor entrada PID temperatura TAQ
PVTempTAQ := TT302.TT01;

// NETWORK 4
//   PIDTT1: Bloco PID para controle de temperatura do TAQ
//   ModoTempTAQ: modo PID temperatura TAQ
//   PVTempTAQ: Valor entrada PID temperatura TAQ
//   SetPointTempTAQ: Set point PID temperatura TAQ
//   ValorManualTempTAQ: Valor manual PID temperatura TAQ
//   TTAQMAX: Temperatura máxima para o TAQ
//   TTAQMIN: Temperatura minima para o TAQ
//   GanhoTempTAQ: Ganho PID temperatura TAQ
//   TITempTAQ: Ti PID temperatura TAQ
//   TDTempTAQ: Td PID temperatura TAQ
//   STPIDTT1: inidicação de saturação na MV
//   OVPIDTT1: indicação de overflow no termo integral
//   TTC01: Comando para a resistência do TAQ
PIDTT1(
    modo := ModoTempTAQ,
    PV := PVTempTAQ,
    SP := SetPointTempTAQ,
    VManual := ValorManualTempTAQ,
    LMAX := TTAQMAX,
    LMIN := TTAQMIN,
    KP := GanhoTempTAQ,
    Ti := TITempTAQ,
    Td := TDTempTAQ,
    satura => STPIDTT1,
    TiOver => OVPIDTT1); // PIDCONTROL
TTC01 := PIDTT1.MV;

// NETWORK 5
//   AO_01: bloco de saida da valvula LCV1 que corresponde a valvula de entrada do TAQ
//   TTC01: Comando para a resistência do TAQ
//   Var_processo.TC_TAQ: comando para resistência de aquecimento do TAQ (TTC01)
AO_01(INPUT := TTC01); // AO
Var_processo.TC_TAQ := AO_01.OUTPUT;

// NETWORK 6

END_PROGRAM
